// TIA Portal V20 export
TYPE "UDT_Service_ServParameter"
   STRUCT
      Analog : Array[0..31] of "UDT_MTP_AnaServParam";
      Digital : Array[0..7] of "UDT_MTP_DIntServParam";
      Binary : Array[0..31] of "UDT_MTP_BinServParam";
      "String" : Array[0..7] of "UDT_MTP_StringServParam";
   END_STRUCT;
END_TYPE
